// Mitsubishi GX Works2 project: project Group N 6 TankUpdate   PLC: FX3G

// global labels: Global1
VAR_GLOBAL
  StorageCounter AT D2000 : REAL;
  ZeroForD1300 AT E0.0 : REAL;
  ZeroFor8282 AT K0 : INT;
  AnalogOutputDisplay AT D8282 : INT;
  DayStart AT X007 : BOOL;
  CurrentRaspberry AT D1120 : REAL;
  CurrentLemon AT D1140 : REAL;
  InitialStabilizer AT D1150 : REAL;
  CurrentStabilizer AT D1160 : REAL;
  InitialGummy AT D1170 : REAL;
  CurrentGummy AT D1180 : REAL;
  RCheckNorm AT M10 : BOOL;
END_VAR
VAR_GLOBAL CONSTANT
  RLimitMin280 : REAL := 280;
END_VAR
VAR_GLOBAL
  LCheckNorm AT M11 : BOOL;
END_VAR
VAR_GLOBAL CONSTANT
  SLimitMin105 : REAL := 105;
  LLimitMin455 : REAL := 455;
END_VAR
VAR_GLOBAL
  SCheckNorm AT M12 : BOOL;
END_VAR
VAR_GLOBAL CONSTANT
  GLimitMin28 : REAL := 28;
END_VAR
VAR_GLOBAL
  GCheckNorm AT M13 : BOOL;
  TypeAnalogValue AT D7000 : REAL;
  IinitialLemon AT D1130 : REAL;
  IinitialRaspberry AT D1100 : REAL;
  Value400 AT E400.0 : REAL;
  MinNormValue AT E0.0 : REAL;
  MaxNormValue AT E5.0 : REAL;
  MinPinukValue AT E6.0 : REAL;
  MaxPinukValue AT E10.0 : REAL;
  IsNorm AT M1 : BOOL;
  IsPinuk AT M2 : BOOL;
  NormInventory AT M19 : BOOL;
  RCheckPinuk AT M30 : BOOL;
  LCheckPinuk AT M31 : BOOL;
  SCheckPinuk AT M32 : BOOL;
  GCheckPinuk AT M33 : BOOL;
  PinukInventory AT M39 : BOOL;
  StartIceCreamProcess AT X001 : BOOL;
  NoInventory AT M99 : BOOL;
  Emergency AT X005 : BOOL;
  StillWorking AT Y007 : BOOL;
  DayIsON AT Y007 : BOOL;
  Sec5 AT K500 : INT;
  IceCreamInMaking AT Y000 : BOOL;
  Sec8 AT K800 : INT;
  FinishIceCream AT M190 : BOOL;
  Temp10 AT X003 : BOOL;
  IsCooling AT Y002 : BOOL;
  CurrentContainerL AT D7994 : REAL;
  InitialContainerR AT E0.0 : REAL;
  InitialContainerL AT E0.0 : REAL;
  CurrentlContainerR AT D7990 : REAL;
  InitialCoolTankR AT E0.0 : REAL;
  InitialCoolTankL AT E0.0 : REAL;
  MixingTankNormal AT D2200 : REAL;
  InitialMixTankNorm AT E0.0 : REAL;
  InitialMixTankPinuk AT E0.0 : REAL;
  MixingTankPinuk AT D2300 : REAL;
  CoolingTankR AT D2050 : REAL;
  CoolingTankL AT D2100 : REAL;
  PinukValue560 AT K560 : INT;
  NormValueR490 AT K490 : INT;
  PinukValue700 AT K700 : INT;
  T8Sec AT TC210 : BOOL;
  T5Sec AT TC200 : BOOL;
  Timer5Sec AT TS200 : BOOL;
  Timer8Sec AT TS210 : BOOL;
  FinishCool AT M200 : BOOL;
  GummyNorm28 AT E28.0 : REAL;
  GummyPinuk70 AT E70.0 : REAL;
  MixedNorm868 AT E868.0 : REAL;
  MixedPinuk1330 AT E1330.0 : REAL;
  TimerHivhuvNorm AT TS4 : BOOL;
  HivhuvNorm AT K30 : INT;
  TmerHivhuvPinuk AT TC5 : BOOL;
  HivhuvPinuk AT K50 : INT;
  FinishMix AT M310 : BOOL;
  Hivhuv AT M320 : BOOL;
  TimerHivhuv AT TS2 : BOOL;
  FirstHivhuv AT Y005 : BOOL;
  TimerHivhuvY5 AT TC2 : BOOL;
  LightTime AT K5 : INT;
  TmerHivhuv2Y6 AT TC3 : BOOL;
  TimerHivhuv2 AT TS3 : BOOL;
  SecondHivhuv AT Y006 : BOOL;
  TimerHivhuvNormS AT TS4 : BOOL;
  TimerHivhuvPinukS AT TS5 : BOOL;
  SinglePackage AT E1.0 : REAL;
  DisplayPackges AT M330 : BOOL;
  MulBy40 AT K40 : INT;
  AnalogInputFirst AT D8280 : INT;
  TypeAnalog AT D7020 : REAL;
  FinishInputAnalog AT M21 : BOOL;
  ZeroForD700 AT E0.0 : REAL;
  StartCooling AT X002 : BOOL;
END_VAR
VAR_GLOBAL CONSTANT
  RLimitMin385 : REAL := 385;
  LLimitMin665 : REAL := 665;
  SLimitMin210 : REAL := 210;
  GLimitMin70 : REAL := 70;
  NormValueR350 : REAL := 350;
  PinukValueR560 : REAL := 560;
  NormValueL490 : REAL := 490;
  PinukValueL700 : REAL := 700;
END_VAR

// task Task_01 (event TRUE, interval 0, priority 31): POU_01

PROGRAM POU_01
(* structured ladder/FBD written out as ST: instructions are called as NAME(EN, inputs, outputs); _pN, _eN, _tN stand for wires *)
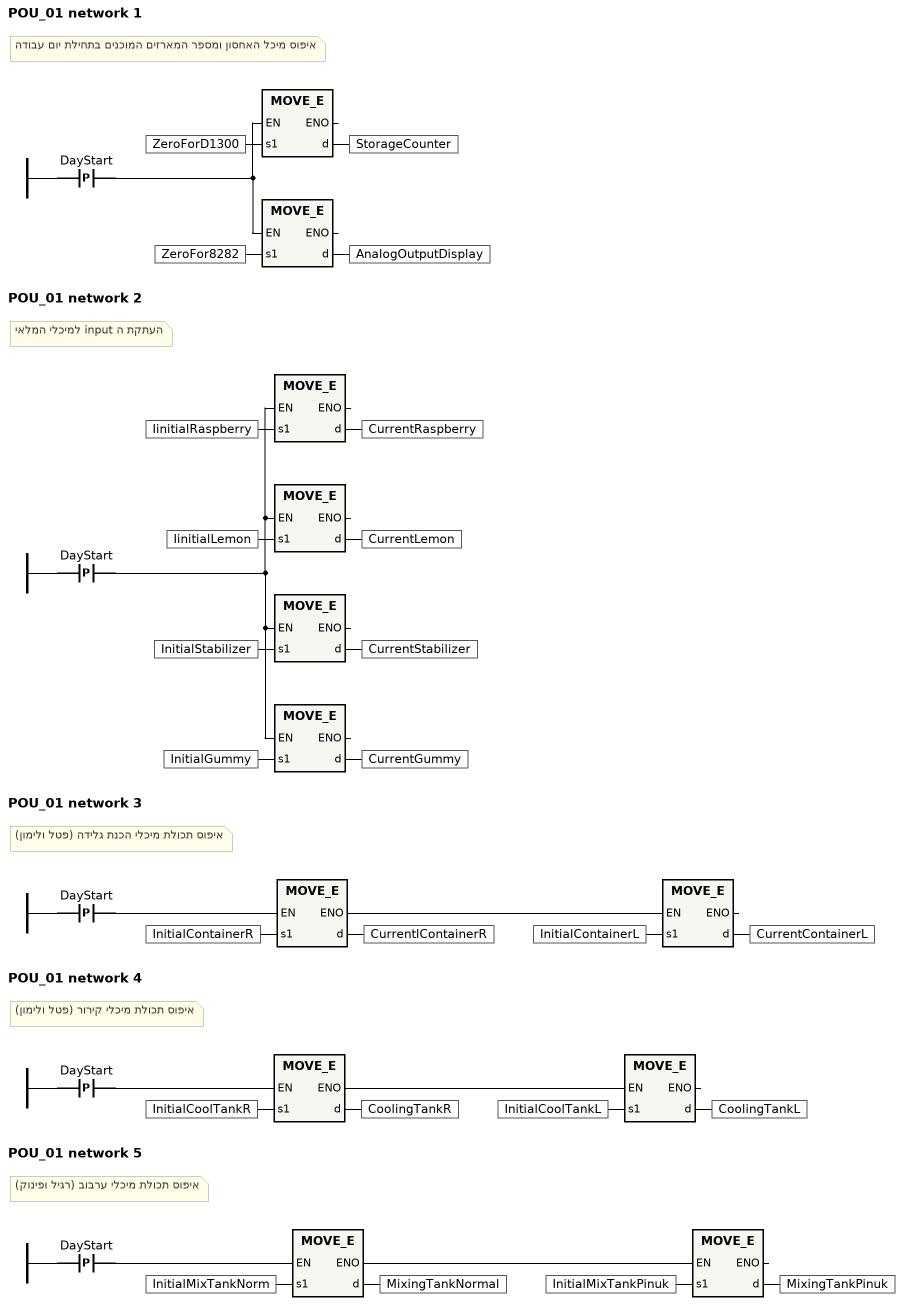
(* network 1 *)
(* איפוס מיכל האחסון ומספר המארזים המוכנים בתחילת יום עבודה *)
_p1 := LDP(TRUE, DayStart);
MOVE_E(_p1, ZeroForD1300, StorageCounter);
MOVE_E(_p1, ZeroFor8282, AnalogOutputDisplay);
(* network 2 *)
(* העתקת ה input למיכלי המלאי *)
_p1 := LDP(TRUE, DayStart);
MOVE_E(_p1, IinitialRaspberry, CurrentRaspberry);
MOVE_E(_p1, IinitialLemon, CurrentLemon);
MOVE_E(_p1, InitialStabilizer, CurrentStabilizer);
MOVE_E(_p1, InitialGummy, CurrentGummy);
(* network 3 *)
(* איפוס תכולת מיכלי הכנת גלידה (פטל ולימון) *)
_e1 := MOVE_E(LDP(TRUE, DayStart), InitialContainerR, CurrentlContainerR);
MOVE_E(_e1, InitialContainerL, CurrentContainerL);
(* network 4 *)
(* איפוס תכולת מיכלי קירור (פטל ולימון) *)
_e1 := MOVE_E(LDP(TRUE, DayStart), InitialCoolTankR, CoolingTankR);
MOVE_E(_e1, InitialCoolTankL, CoolingTankL);
(* network 5 *)
(* איפוס תכולת מיכלי ערבוב (רגיל ופינוק) *)
_e1 := MOVE_E(LDP(TRUE, DayStart), InitialMixTankNorm, MixingTankNormal);
MOVE_E(_e1, InitialMixTankPinuk, MixingTankPinuk);
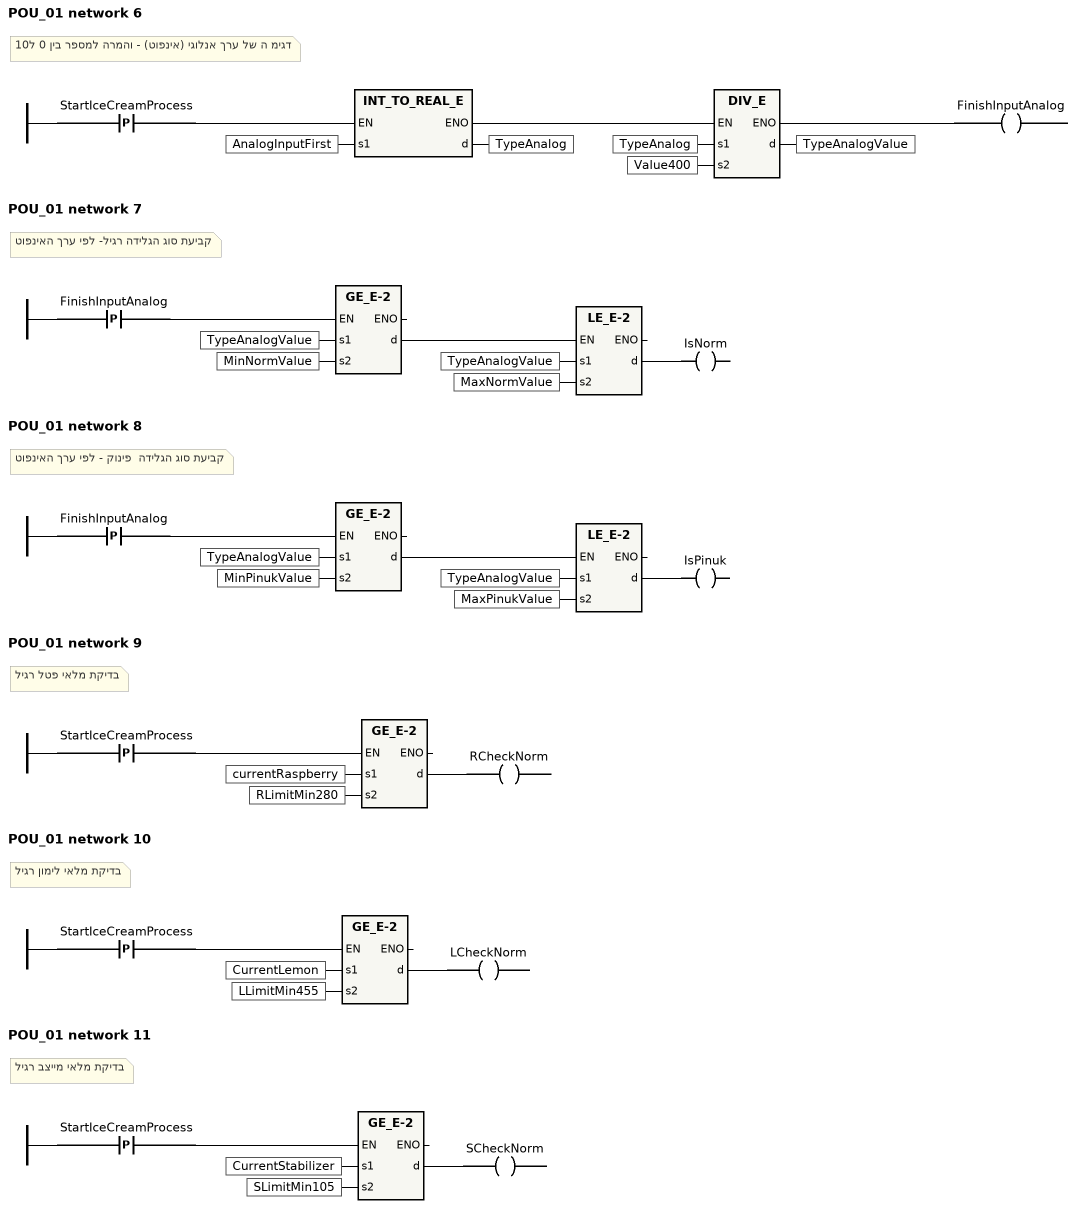
(* network 6 *)
(* דגימ ה של ערך אנלוגי (אינפוט) - והמרה למספר בין 0 ל10 *)
_e1 := INT_TO_REAL_E(LDP(TRUE, StartIceCreamProcess), AnalogInputFirst, TypeAnalog);
_e2 := DIV_E(_e1, TypeAnalog, Value400, TypeAnalogValue);
FinishInputAnalog := _e2;
(* network 7 *)
(* קביעת סוג הגלידה רגיל- לפי ערך האינפוט *)
GE_E(LDP(TRUE, FinishInputAnalog), TypeAnalogValue, MinNormValue, _t1);
LE_E(_t1, TypeAnalogValue, MaxNormValue, _t2);
IsNorm := _t2;
(* network 8 *)
(* קביעת סוג הגלידה  פינוק - לפי ערך האינפוט *)
GE_E(LDP(TRUE, FinishInputAnalog), TypeAnalogValue, MinPinukValue, _t1);
LE_E(_t1, TypeAnalogValue, MaxPinukValue, _t2);
IsPinuk := _t2;
(* network 9 *)
(* בדיקת מלאי פטל רגיל *)
GE_E(LDP(TRUE, StartIceCreamProcess), currentRaspberry, RLimitMin280, _t1);
RCheckNorm := _t1;
(* network 10 *)
(* בדיקת מלאי לימון רגיל *)
GE_E(LDP(TRUE, StartIceCreamProcess), CurrentLemon, LLimitMin455, _t1);
LCheckNorm := _t1;
(* network 11 *)
(* בדיקת מלאי מייצב רגיל *)
GE_E(LDP(TRUE, StartIceCreamProcess), CurrentStabilizer, SLimitMin105, _t1);
SCheckNorm := _t1;
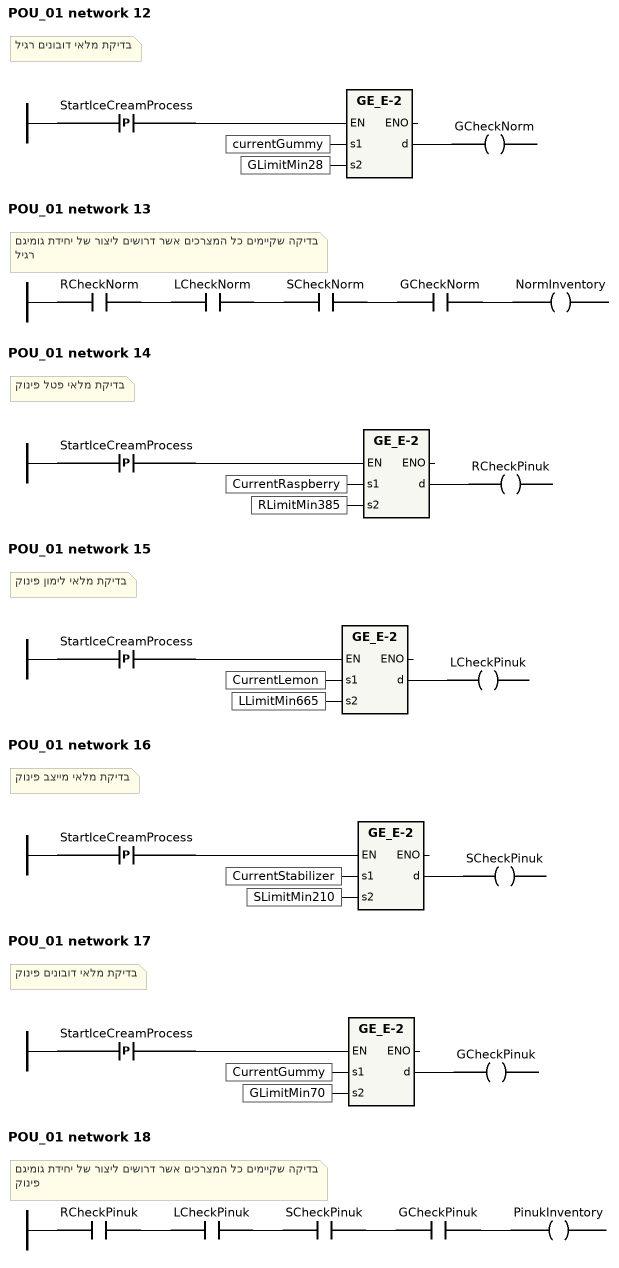
(* network 12 *)
(* בדיקת מלאי דובונים רגיל *)
GE_E(LDP(TRUE, StartIceCreamProcess), currentGummy, GLimitMin28, _t1);
GCheckNorm := _t1;
(* network 13 *)
(* בדיקה שקיימים כל המצרכים אשר דרושים ליצור של יחידת גומיגם רגיל *)
NormInventory := RCheckNorm AND LCheckNorm AND SCheckNorm AND GCheckNorm;
(* network 14 *)
(* בדיקת מלאי פטל פינוק *)
GE_E(LDP(TRUE, StartIceCreamProcess), CurrentRaspberry, RLimitMin385, _t1);
RCheckPinuk := _t1;
(* network 15 *)
(* בדיקת מלאי לימון פינוק *)
GE_E(LDP(TRUE, StartIceCreamProcess), CurrentLemon, LLimitMin665, _t1);
LCheckPinuk := _t1;
(* network 16 *)
(* בדיקת מלאי מייצב פינוק *)
GE_E(LDP(TRUE, StartIceCreamProcess), CurrentStabilizer, SLimitMin210, _t1);
SCheckPinuk := _t1;
(* network 17 *)
(* בדיקת מלאי דובונים פינוק *)
GE_E(LDP(TRUE, StartIceCreamProcess), CurrentGummy, GLimitMin70, _t1);
GCheckPinuk := _t1;
(* network 18 *)
(* בדיקה שקיימים כל המצרכים אשר דרושים ליצור של יחידת גומיגם פינוק *)
PinukInventory := RCheckPinuk AND LCheckPinuk AND SCheckPinuk AND GCheckPinuk;
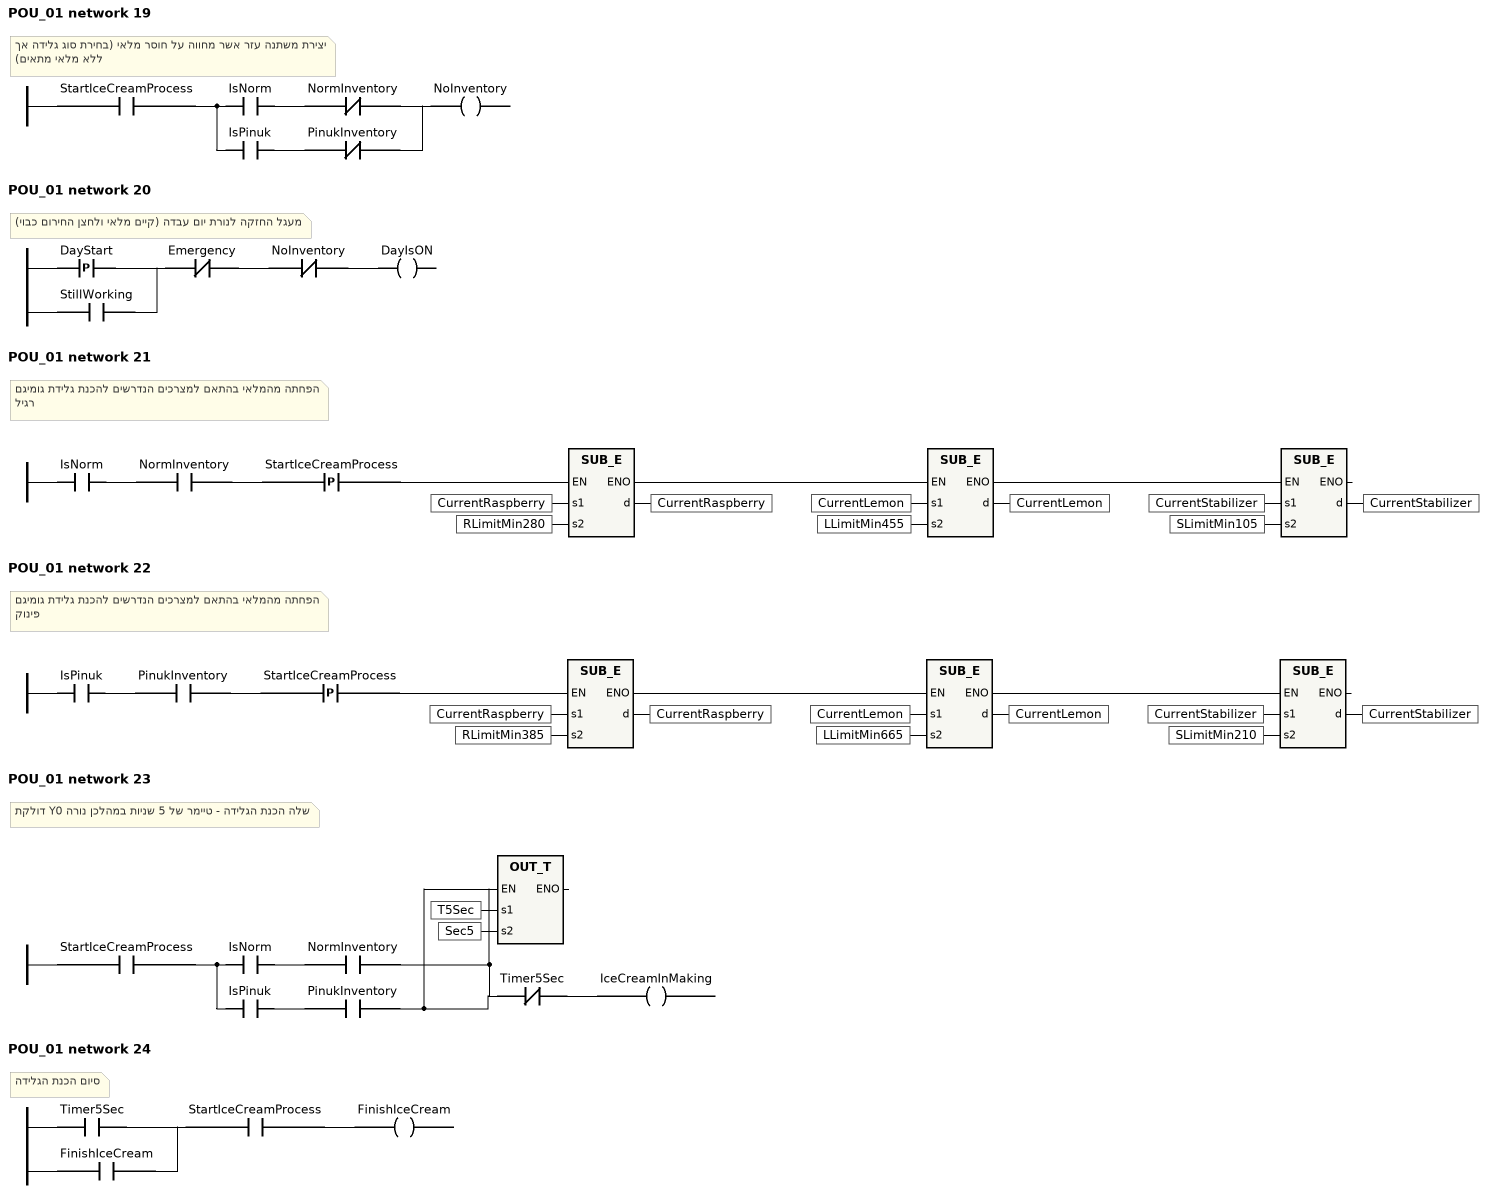
(* network 19 *)
(* יצירת משתנה עזר אשר מחווה על חוסר מלאי (בחירת סוג גלידה אך ללא מלאי מתאים) *)
NoInventory := (StartIceCreamProcess AND IsNorm AND NOT NormInventory) OR (StartIceCreamProcess AND IsPinuk AND NOT PinukInventory);
(* network 20 *)
(* מעגל החזקה לנורת יום עבדה (קיים מלאי ולחצן החירום כבוי) *)
DayIsON := ((LDP(TRUE, DayStart) OR StillWorking) AND NOT Emergency) AND NOT NoInventory;
(* network 21 *)
(* הפחתה מהמלאי בהתאם למצרכים הנדרשים להכנת גלידת גומיגם רגיל *)
_e1 := SUB_E(IsNorm AND NormInventory AND LDP(TRUE, StartIceCreamProcess), CurrentRaspberry, RLimitMin280, CurrentRaspberry);
_e2 := SUB_E(_e1, CurrentLemon, LLimitMin455, CurrentLemon);
SUB_E(_e2, CurrentStabilizer, SLimitMin105, CurrentStabilizer);
(* network 22 *)
(* הפחתה מהמלאי בהתאם למצרכים הנדרשים להכנת גלידת גומיגם פינוק *)
_e1 := SUB_E(IsPinuk AND PinukInventory AND LDP(TRUE, StartIceCreamProcess), CurrentRaspberry, RLimitMin385, CurrentRaspberry);
_e2 := SUB_E(_e1, CurrentLemon, LLimitMin665, CurrentLemon);
SUB_E(_e2, CurrentStabilizer, SLimitMin210, CurrentStabilizer);
(* network 23 *)
(* שלה הכנת הגלידה - טיימר של 5 שניות במהלכן נורה Y0 דולקת *)
_p1 := (StartIceCreamProcess AND IsNorm AND NormInventory) OR (StartIceCreamProcess AND IsPinuk AND PinukInventory);
OUT_T(_p1, T5Sec, Sec5);
IceCreamInMaking := _p1 AND NOT Timer5Sec;
(* network 24 *)
(* סיום הכנת הגלידה *)
FinishIceCream := (Timer5Sec OR FinishIceCream) AND StartIceCreamProcess;
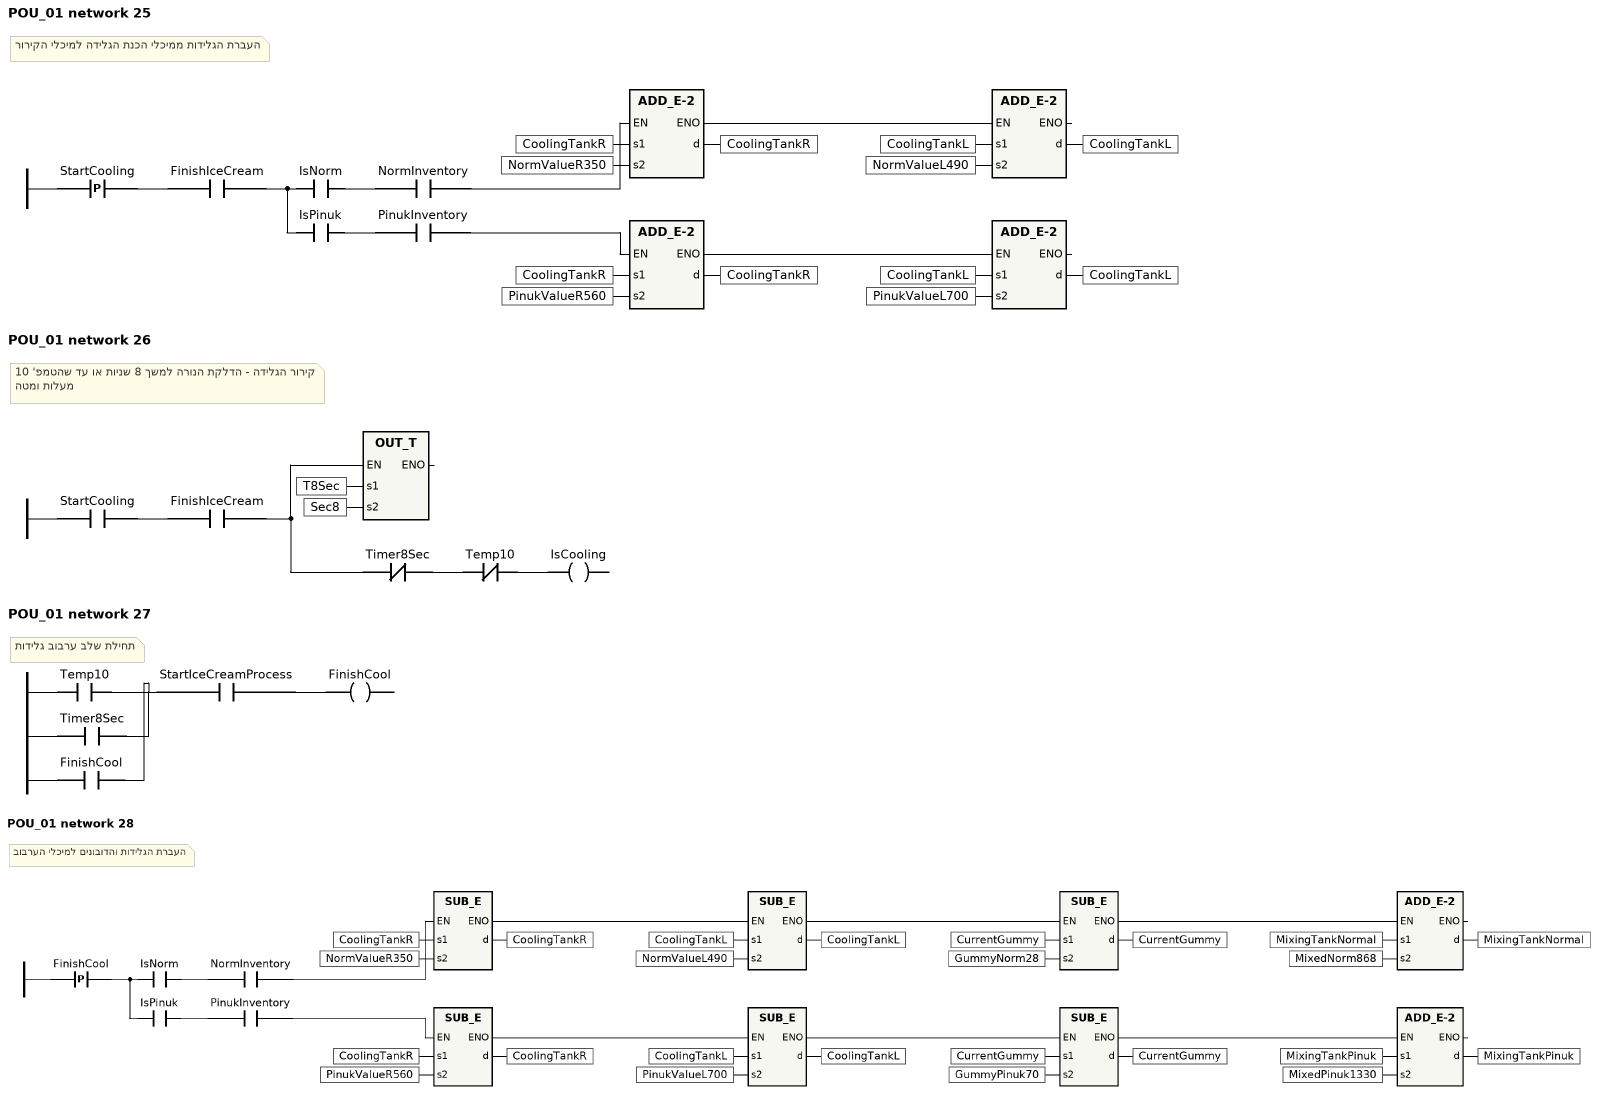
(* network 25 *)
(* העברת הגלידות ממיכלי הכנת הגלידה למיכלי הקירור *)
_p1 := LDP(TRUE, StartCooling) AND FinishIceCream;
_e2 := ADD_E(_p1 AND IsNorm AND NormInventory, CoolingTankR, NormValueR350, CoolingTankR);
ADD_E(_e2, CoolingTankL, NormValueL490, CoolingTankL);
_e3 := ADD_E(_p1 AND IsPinuk AND PinukInventory, CoolingTankR, PinukValueR560, CoolingTankR);
ADD_E(_e3, CoolingTankL, PinukValueL700, CoolingTankL);
(* network 26 *)
(* קירור הגלידה - הדלקת הנורה למשך 8 שניות או עד שהטמפ' 10 מעלות ומטה *)
_p1 := StartCooling AND FinishIceCream;
OUT_T(_p1, T8Sec, Sec8);
IsCooling := _p1 AND NOT Timer8Sec AND NOT Temp10;
(* network 27 *)
(* תחילת שלב ערבוב גלידות *)
FinishCool := (Temp10 OR Timer8Sec OR FinishCool) AND StartIceCreamProcess;
(* network 28 *)
(* העברת הגלידות והדובונים למיכלי הערבוב *)
_p1 := LDP(TRUE, FinishCool);
_e2 := SUB_E(_p1 AND IsNorm AND NormInventory, CoolingTankR, NormValueR350, CoolingTankR);
_e3 := SUB_E(_e2, CoolingTankL, NormValueL490, CoolingTankL);
_e4 := SUB_E(_e3, CurrentGummy, GummyNorm28, CurrentGummy);
ADD_E(_e4, MixingTankNormal, MixedNorm868, MixingTankNormal);
_e5 := SUB_E(_p1 AND IsPinuk AND PinukInventory, CoolingTankR, PinukValueR560, CoolingTankR);
_e6 := SUB_E(_e5, CoolingTankL, PinukValueL700, CoolingTankL);
_e7 := SUB_E(_e6, CurrentGummy, GummyPinuk70, CurrentGummy);
ADD_E(_e7, MixingTankPinuk, MixedPinuk1330, MixingTankPinuk);
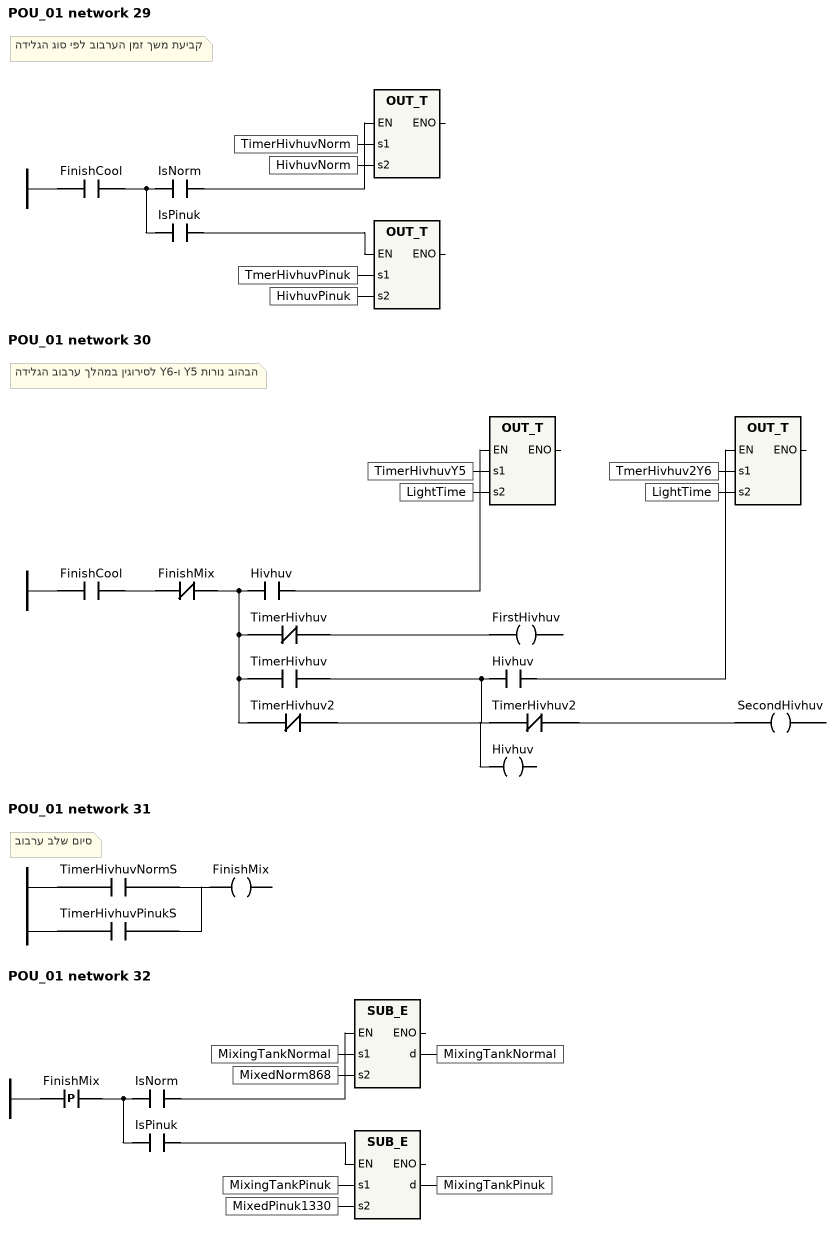
(* network 29 *)
(* קביעת משך זמן הערבוב לפי סוג הגלידה *)
OUT_T(FinishCool AND IsNorm, TimerHivhuvNorm, HivhuvNorm);
OUT_T(FinishCool AND IsPinuk, TmerHivhuvPinuk, HivhuvPinuk);
(* network 30 *)
(* הבהוב נורות Y5 ו-Y6 לסירוגין במהלך ערבוב הגלידה *)
_p1 := FinishCool AND NOT FinishMix;
OUT_T(_p1 AND Hivhuv, TimerHivhuvY5, LightTime);
FirstHivhuv := _p1 AND NOT TimerHivhuv;
_p2 := _p1 AND TimerHivhuv;
OUT_T(_p2 AND Hivhuv, TmerHivhuv2Y6, LightTime);
SecondHivhuv := _p2 AND NOT TimerHivhuv2;
Hivhuv := _p1 AND NOT TimerHivhuv2;
(* network 31 *)
(* סיום שלב ערבוב *)
FinishMix := TimerHivhuvNormS OR TimerHivhuvPinukS;
(* network 32 *)
_p1 := LDP(TRUE, FinishMix);
SUB_E(_p1 AND IsNorm, MixingTankNormal, MixedNorm868, MixingTankNormal);
SUB_E(_p1 AND IsPinuk, MixingTankPinuk, MixedPinuk1330, MixingTankPinuk);
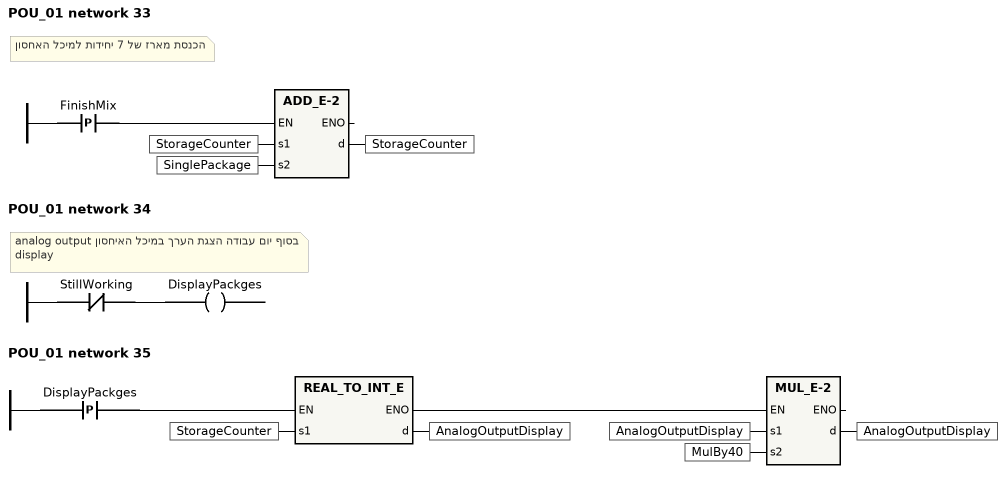
(* network 33 *)
(* הכנסת מארז של 7 יחידות למיכל האחסון *)
ADD_E(LDP(TRUE, FinishMix), StorageCounter, SinglePackage, StorageCounter);
(* network 34 *)
(* בסוף יום עבודה הצגת הערך במיכל האיחסון analog output display *)
DisplayPackges := NOT StillWorking;
(* network 35 *)
_e1 := REAL_TO_INT_E(LDP(TRUE, DisplayPackges), StorageCounter, AnalogOutputDisplay);
MUL_E(_e1, AnalogOutputDisplay, MulBy40, AnalogOutputDisplay);
END_PROGRAM
